
// ===== library: MasterCopy "Data_block_1" =====

DATA_BLOCK "Data_block_1"   // DB1
{ S7_Optimized_Access := 'TRUE' }
VERSION : 0.1
   VAR
      START : Bool;
      EXTEND : Bool;
      RETRACT : Bool;
      "POSITION CONTROL" : Real;
      PISTON_EXTEND : Bool;
      PISTON_RETRACT : Bool;
   END_VAR
BEGIN
END_DATA_BLOCK